{attribute 'GeneratedUsingTerminal: BK1250-0000-0016'}
{attribute addProperty BoxType "BK1250-0000-0016"}
{attribute addProperty Id "Term_396_KL1002KL1002_BB38DA8F0"}
{attribute addProperty CRC "1598977783"}
{attribute addProperty Size "0"}
TYPE A_0015_BK1250_0000_0016_5F4E76F7 EXTENDS BK1250_A2FCADE7 :
STRUCT
	{attribute addProperty Name "Term_396_KL1002"}
	Term_396_KL1002 : KL1002_BB38DA8F;
END_STRUCT
END_TYPE

(* stored: Version 1.2.0.0, ProductVersion 3.1.4024.9
   DUT A_0015_BK1250_0000_0016_5F4E76F7: Id {ce4b1835-1fb9-4a99-89a2-da739cf0a49c} *)
